{attribute 'GeneratedUsingTerminal: EP6224-0042-0016'}
{attribute addProperty BoxType "EP6224-0042-0016"}
{attribute addProperty Id "EtcSlaveTerminalBaseModule_1_DeviceState_Inputs_DeviceModule_1_DeviceState_Inputs_Device_5322301C2Module_2_DeviceState_InputsModule_2_DeviceState_Inputs_BD6C70354Module_7_Digital_InputsModule_7_Digital_Inputs_DAAE149B8WcStateAT %I*WcState_9091E0EB2InfoDataAT %I*InfoData_90184F0C16"}
{attribute addProperty CRC "2676080768"}
{attribute addProperty Size "32"}
TYPE EP6224_9F81C080 EXTENDS EtcSlaveTerminalBase :
STRUCT
	{attribute addProperty Name "Module_1_DeviceState_Inputs_Device"}
	Module_1_DeviceState_Inputs_Device : Module_1_DeviceState_Inputs_Device_5322301C;
	{attribute addProperty Name "Module_2_DeviceState_Inputs"}
	Module_2_DeviceState_Inputs : Module_2_DeviceState_Inputs_BD6C7035;
	{attribute addProperty Name "Module_7_Digital_Inputs"}
	Module_7_Digital_Inputs : Module_7_Digital_Inputs_DAAE149B;
	{attribute addProperty Name "WcState"}
	WcState : WcState_9091E0EB;
	{attribute addProperty Name "InfoData"}
	InfoData : InfoData_90184F0C;
END_STRUCT
END_TYPE

(* stored: Version 1.2.0.0, ProductVersion 3.1.4024.9
   DUT EP6224_9F81C080: Id {8afdaac8-3208-4d55-a295-8158941ddcfa} *)
